// Brief: Setup Arm Adjust
FUNCTION_BLOCK PUBLIC FB_SetupCtrlAutoAdjust EXTENDS FB_SetupArmCtrlBase
VAR_INPUT
END_VAR
VAR_OUTPUT
END_VAR
VAR
END_VAR

METHOD PUBLIC init : BOOL
VAR_IN_OUT CONSTANT
	i_setupArm	:FB_SetupArm;
END_VAR
VAR_IN_OUT 
	r_setupArmCtrlCmd :ST_SetupArmCtrlCmds;
END_VAR
SUPER^.Init(i_setupArm,r_setupArmCtrlCmd);
END_METHOD

END_FUNCTION_BLOCK

(* stored: Version 1.1.0.1, ProductVersion 3.1.4024.12
   POU FB_SetupCtrlAutoAdjust: Id {53032ea5-b008-491f-a641-5219ef32615c}, SpecialFunc None
   Method init: Id {dd68468f-e9b8-4053-9776-4b6e1ffcee16} *)
